TYPE TYP_VAC_GEN_HW_IN :
STRUCT
	ReachedVac AT %I* : BOOL;
END_STRUCT
END_TYPE

(* stored: Version 1.1.0.1, ProductVersion 3.1.4024.12
   DUT TYP_VAC_GEN_HW_IN: Id {6aedd216-9f6b-4b52-8dbf-0b0a27b66307} *)
